{attribute 'qualified_only'}
VAR_GLOBAL
    _basicRunnerTests : fbBasicRunnerTests;
    _recorderRunnerTests : fbRecorderRunnerTests;
END_VAR

(* stored: Version 1.1.0.1, ProductVersion 3.1.4024.4
   GVL Tests: Id {e5858b03-19b3-430c-8807-95ad52fea761} *)
